Staubli VAL3: getVelocity.pgx

public program getVelocity(string& x_sItem[], num& x_nVelocity[])
  local num l_nSize
begin
  call getSize(l_nSize)
  for i=0 to l_nSize
    call get(l_sItem,i)
    if l_sItem==x_sItem
      x_nVelocity=nVelocity[i]
      return
      //go back
    endIf
  endFor
end
